KUKA KRL program: Safety_Position.src, Safety_Position.dat

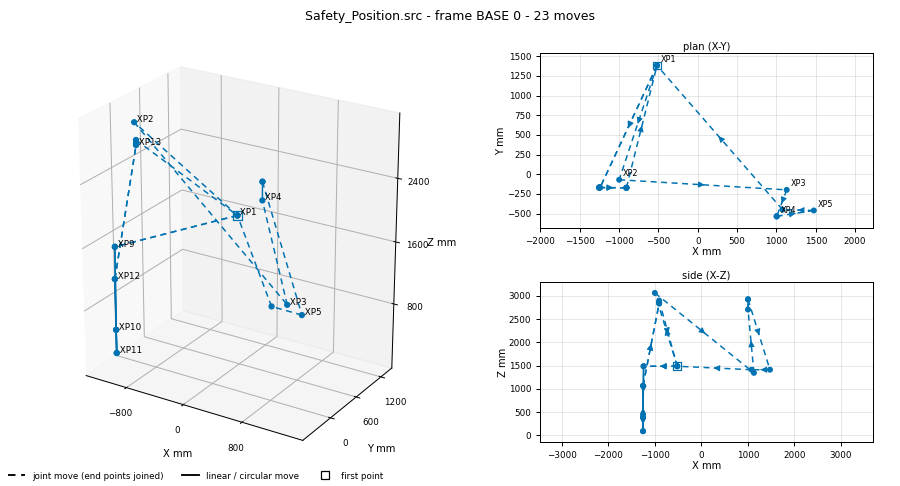
[picture p0: tool path of Safety_Position.src in frame BASE 0, 23 of 23 moves have a stored position in this frame; points joined in program order, loops and branches not executed]
--- Safety_Position.src ---
&ACCESS RVP8
&REL 86
&COMMENT Safety Position
&PARAM DISKPATH = KRC:\R1\Program\Safety Programs
DEF SAFETY_POSITION(DIRECTION :IN,AREA_NR :IN,TYPE_NR :IN )
;FOLD INI
  INT DIRECTION
  INT AREA_NR
  INT TYPE_NR
  decl KrlMsg_T msg
  decl KrlMsgPar_T par[3]
  decl KrlMsgOpt_T opt
  INT nHandle

  IF (DIRECTION>2) OR (DIRECTION<1) THEN
    REPEAT
      msg = {modul[] "Safety Position", nr 1, msg_txt[] "Direction Number Not Valid"}

			opt = {vl_stop true, clear_p_reset true, clear_p_SAW false, log_to_DB false}

			nHandle = Set_KrlMsg(#notify, msg, par[], opt)
      HALT
    UNTIL (DIRECTION<3) AND (DIRECTION>0)
  ENDIF
  IF (AREA_NR>8) OR (AREA_NR<1) THEN
    REPEAT
      msg = {modul[] "Safety Position", nr 2, msg_txt[] "Area Number Not Valid"}

			opt = {vl_stop true, clear_p_reset true, clear_p_SAW false, log_to_DB false}

			nHandle = Set_KrlMsg(#notify, msg, par[], opt)
      HALT
    UNTIL (AREA_NR<9) AND (AREA_NR>0)
  ENDIF
  IF (TYPE_NR>8) OR (TYPE_NR<1) THEN
    REPEAT
  	  msg = {modul[] "Safety Position", nr 1, msg_txt[] "Type Number Not Valid"}

			opt = {vl_stop true, clear_p_reset true, clear_p_SAW false, log_to_DB false}

			nHandle = Set_KrlMsg(#notify, msg, par[], opt)
      HALT
    UNTIL (TYPE_NR<9) AND (TYPE_NR>0)
  ENDIF
  ;ENDFOLD
;===================================================
; MODEL     :CX482
; IE GROUP  :PHEV
; STATION   :110
; ROBOT     :110R1
; FUNCTION  : Safety Position
;================================================

SWITCH AREA_NR

CASE 1  ;AREA 1

  SWITCH TYPE_NR

  CASE 1  ;Area 1 - Safety Position 1
    SWITCH DIRECTION
    CASE 1
    ;Teach here positions from wait area to safety position
;FOLD PTP P1 CONT Vel=50 % PDAT1 Tool[5] Base[0];%{PE}%R 8.3.48,%MKUKATPBASIS,%CMOVE,%VPTP,%P 1:PTP, 2:P1, 3:C_DIS, 5:50, 7:PDAT1
$BWDSTART=FALSE
PDAT_ACT=PPDAT1
FDAT_ACT=FP1
BAS(#PTP_PARAMS,50)
PTP XP1 C_DIS
;ENDFOLD
;FOLD PTP P2 Vel=50 % PDAT2 Tool[5] Base[0];%{PE}%R 8.3.48,%MKUKATPBASIS,%CMOVE,%VPTP,%P 1:PTP, 2:P2, 3:, 5:50, 7:PDAT2
$BWDSTART=FALSE
PDAT_ACT=PPDAT2
FDAT_ACT=FP2
BAS(#PTP_PARAMS,50)
PTP XP2
;ENDFOLD
    ;check robot movement for collision with other robots
    CASE 2
    ;Teach here positions from safety position to wait area
;FOLD PTP P3 CONT Vel=100 % PDAT3 Tool[5] Base[0];%{PE}%R 8.3.48,%MKUKATPBASIS,%CMOVE,%VPTP,%P 1:PTP, 2:P3, 3:C_DIS, 5:100, 7:PDAT3
$BWDSTART=FALSE
PDAT_ACT=PPDAT3
FDAT_ACT=FP3
BAS(#PTP_PARAMS,100)
PTP XP3 C_DIS
;ENDFOLD
;FOLD PTP P4 Vel=100 % PDAT4 Tool[5] Base[0];%{PE}%R 8.3.48,%MKUKATPBASIS,%CMOVE,%VPTP,%P 1:PTP, 2:P4, 3:, 5:100, 7:PDAT4
$BWDSTART=FALSE
PDAT_ACT=PPDAT4
FDAT_ACT=FP4
BAS(#PTP_PARAMS,100)
PTP XP4
;ENDFOLD
    ;check robot movement for collision with other robots
    ENDSWITCH

  CASE 2  ;Area 1 - Safety Position 2

    SWITCH DIRECTION
    CASE 1
lin_rel {z 220}
lin_rel {b 20}
;FOLD PTP P5 CONT Vel=100 % PDAT5 Tool[5] Base[0];%{PE}%R 8.3.48,%MKUKATPBASIS,%CMOVE,%VPTP,%P 1:PTP, 2:P5, 3:C_DIS, 5:100, 7:PDAT5
$BWDSTART=FALSE
PDAT_ACT=PPDAT5
FDAT_ACT=FP5
BAS(#PTP_PARAMS,100)
PTP XP5 C_DIS
;ENDFOLD
;FOLD PTP P7 CONT Vel=100 % PDAT7 Tool[5] Base[0];%{PE}%R 8.3.48,%MKUKATPBASIS,%CMOVE,%VPTP,%P 1:PTP, 2:P7, 3:C_DIS, 5:100, 7:PDAT7
$BWDSTART=FALSE
PDAT_ACT=PPDAT7
FDAT_ACT=FP7
BAS(#PTP_PARAMS,100)
PTP XP7 C_DIS
;ENDFOLD
;FOLD PTP P6 CONT Vel=100 % PDAT6 Tool[5] Base[0];%{PE}%R 8.3.48,%MKUKATPBASIS,%CMOVE,%VPTP,%P 1:PTP, 2:P6, 3:C_DIS, 5:100, 7:PDAT6
$BWDSTART=FALSE
PDAT_ACT=PPDAT6
FDAT_ACT=FP6
BAS(#PTP_PARAMS,100)
PTP XP6 C_DIS
;ENDFOLD
;FOLD PTP P9 CONT Vel=100 % PDAT9 Tool[5] Base[0];%{PE}%R 8.3.48,%MKUKATPBASIS,%CMOVE,%VPTP,%P 1:PTP, 2:P9, 3:C_DIS, 5:100, 7:PDAT9
$BWDSTART=FALSE
PDAT_ACT=PPDAT9
FDAT_ACT=FP9
BAS(#PTP_PARAMS,100)
PTP XP9 C_DIS
;ENDFOLD
;FOLD LIN P10 CONT Vel=2 m/s CPDAT1 Tool[5] Base[0];%{PE}%R 8.3.48,%MKUKATPBASIS,%CMOVE,%VLIN,%P 1:LIN, 2:P10, 3:C_DIS C_DIS, 5:2, 7:CPDAT1
$BWDSTART=FALSE
LDAT_ACT=LCPDAT1
FDAT_ACT=FP10
BAS(#CP_PARAMS,2)
LIN XP10 C_DIS C_DIS
;ENDFOLD
;FOLD LIN P11 Vel=0.5 m/s CPDAT2 Tool[5] Base[0];%{PE}%R 8.3.48,%MKUKATPBASIS,%CMOVE,%VLIN,%P 1:LIN, 2:P11, 3:, 5:0.5, 7:CPDAT2
$BWDSTART=FALSE
LDAT_ACT=LCPDAT2
FDAT_ACT=FP11
BAS(#CP_PARAMS,0.5)
LIN XP11
;ENDFOLD

;abrir gara
cil_bat_reposo()

;FOLD LIN P12 CONT Vel=0.5 m/s CPDAT3 Tool[5] Base[0];%{PE}%R 8.3.48,%MKUKATPBASIS,%CMOVE,%VLIN,%P 1:LIN, 2:P12, 3:C_DIS C_DIS, 5:0.5, 7:CPDAT3
$BWDSTART=FALSE
LDAT_ACT=LCPDAT3
FDAT_ACT=FP12
BAS(#CP_PARAMS,0.5)
LIN XP12 C_DIS C_DIS
;ENDFOLD
;FOLD PTP P13 CONT Vel=100 % PDAT10 Tool[5] Base[0];%{PE}%R 8.3.48,%MKUKATPBASIS,%CMOVE,%VPTP,%P 1:PTP, 2:P13, 3:C_DIS, 5:100, 7:PDAT10
$BWDSTART=FALSE
PDAT_ACT=PPDAT10
FDAT_ACT=FP13
BAS(#PTP_PARAMS,100)
PTP XP13 C_DIS
;ENDFOLD
    ;Teach here positions from waiting area to safety position
    ;check robot movement for collision with other robots
    CASE 2
lin_rel {z 20}
lin_rel {b 20}
lin_rel {z 40}
;FOLD PTP P14 CONT Vel=100 % PDAT11 Tool[5] Base[0];%{PE}%R 8.3.48,%MKUKATPBASIS,%CMOVE,%VPTP,%P 1:PTP, 2:P14, 3:C_DIS, 5:100, 7:PDAT11
$BWDSTART=FALSE
PDAT_ACT=PPDAT11
FDAT_ACT=FP14
BAS(#PTP_PARAMS,100)
PTP XP14 C_DIS
;ENDFOLD
;FOLD PTP P15 CONT Vel=100 % PDAT12 Tool[5] Base[0];%{PE}%R 8.3.48,%MKUKATPBASIS,%CMOVE,%VPTP,%P 1:PTP, 2:P15, 3:C_DIS, 5:100, 7:PDAT12
$BWDSTART=FALSE
PDAT_ACT=PPDAT12
FDAT_ACT=FP15
BAS(#PTP_PARAMS,100)
PTP XP15 C_DIS
;ENDFOLD
;FOLD LIN P16 CONT Vel=0.5 m/s CPDAT4 Tool[5] Base[0];%{PE}%R 8.3.48,%MKUKATPBASIS,%CMOVE,%VLIN,%P 1:LIN, 2:P16, 3:C_DIS C_DIS, 5:0.5, 7:CPDAT4
$BWDSTART=FALSE
LDAT_ACT=LCPDAT4
FDAT_ACT=FP16
BAS(#CP_PARAMS,0.5)
LIN XP16 C_DIS C_DIS
;ENDFOLD
;FOLD LIN P17 Vel=0.5 m/s CPDAT5 Tool[5] Base[0];%{PE}%R 8.3.48,%MKUKATPBASIS,%CMOVE,%VLIN,%P 1:LIN, 2:P17, 3:, 5:0.5, 7:CPDAT5
$BWDSTART=FALSE
LDAT_ACT=LCPDAT5
FDAT_ACT=FP17
BAS(#CP_PARAMS,0.5)
LIN XP17
;ENDFOLD

;abrir gara
cil_bat_reposo()

;FOLD LIN P18 CONT Vel=0.5 m/s CPDAT6 Tool[5] Base[0];%{PE}%R 8.3.48,%MKUKATPBASIS,%CMOVE,%VLIN,%P 1:LIN, 2:P18, 3:C_DIS C_DIS, 5:0.5, 7:CPDAT6
$BWDSTART=FALSE
LDAT_ACT=LCPDAT6
FDAT_ACT=FP18
BAS(#CP_PARAMS,0.5)
LIN XP18 C_DIS C_DIS
;ENDFOLD
;FOLD PTP P19 CONT Vel=100 % PDAT13 Tool[5] Base[0];%{PE}%R 8.3.48,%MKUKATPBASIS,%CMOVE,%VPTP,%P 1:PTP, 2:P19, 3:C_DIS, 5:100, 7:PDAT13
$BWDSTART=FALSE
PDAT_ACT=PPDAT13
FDAT_ACT=FP19
BAS(#PTP_PARAMS,100)
PTP XP19 C_DIS
;ENDFOLD
    ;Teach here positions from safety position to waiting area
    ;check robot movement for collision with other robots
    ENDSWITCH

  CASE 3  ;Area 1 - Safety Position 3

    SWITCH DIRECTION
    CASE 1
    ;Teach here positions from waiting area to safety position
    ;check robot movement for collision with other robots
    CASE 2
    ;Teach here positions from safety position to waiting area
    ;check robot movement for collision with other robots
    ENDSWITCH

  CASE 4  ;Area 1 - Safety Position 4

    SWITCH DIRECTION
    CASE 1 ; From Area Request Position To Safety Position
    ;Teach here positions from waiting area to safety position
    ;check robot movement for collision with other robots
    CASE 2 ; From Safety Position To Area Request Position
    ;Teach here positions from safety position to waiting area
    ;check robot movement for collision with other robots
    ENDSWITCH

  CASE 5  ;Area 1 - Safety Position 5

    SWITCH DIRECTION
    CASE 1
    ;Teach here positions from waiting area to safety position
    ;check robot movement for collision with other robots
    CASE 2
    ;Teach here positions from safety position to waiting area
    ;check robot movement for collision with other robots
    ENDSWITCH

  CASE 6  ;Area 1 - Safety Position 6

    SWITCH DIRECTION
    CASE 1
    ;Teach here positions from waiting area to safety position
    ;check robot movement for collision with other robots
    CASE 2
    ;Teach here positions from safety position to waiting area
    ;check robot movement for collision with other robots
    ENDSWITCH

  CASE 7  ;Area 1 - Safety Position 7

    SWITCH DIRECTION
    CASE 1
    ;Teach here positions from waiting area to safety position
    ;check robot movement for collision with other robots
    CASE 2
    ;Teach here positions from safety position to waiting area
    ;check robot movement for collision with other robots
    ENDSWITCH

  CASE 8  ;Area 1 - Safety Position 8

    SWITCH DIRECTION
    CASE 1
    ;Teach here positions from wait area to safety position
    ;check robot movement for collision with other robots
    CASE 2
    ;Teach here positions from safety position to wait area
    ;check robot movement for collision with other robots
    ENDSWITCH

  ENDSWITCH

;====================================================================

CASE 2  ;AREA 2

  SWITCH TYPE_NR
  CASE 1  ;Area 2 - Safety Position 1

    SWITCH DIRECTION
    CASE 1
    ;Teach here pos from waiting area to safety position
    ;check robot movement for collision with other robots
    CASE 2
    ;Teach here positions from safety pos to waiting area
    ;check robot movement for collision with other robots
    ENDSWITCH

  CASE 2  ;Area 2 - Safety Position 2

    SWITCH DIRECTION
    CASE 1
    ;Teach here positions from waiting area to safety position
    ;check robot movement for collision with other robots
    CASE 2
    ;Teach here positions from safety position to waiting area
    ;check robot movement for collision with other robots
    ENDSWITCH

  CASE 3  ;Area 2 - Safety Position 3

    SWITCH DIRECTION
    CASE 1
    ;Teach here positions from waiting area to safety position
    ;check robot movement for collision with other robots
    CASE 2
    ;Teach here positions from safety position to waiting area
    ;check robot movement for collision with other robots
    ENDSWITCH

  CASE 4  ;Area 2 - Safety Position 4

    SWITCH DIRECTION
	  	CASE 1
    ;Teach here positions from waiting area to safety position
    ;check robot movement for collision with other robots
    CASE 2
    ;Teach here positions from safety position to waiting area
    ;check robot movement for collision with other robots
    ENDSWITCH

  CASE 5  ;Area 2 - Safety Position 5

    SWITCH DIRECTION
    CASE 1
    ;Teach here positions from waiting area to safety position
    ;check robot movement for collision with other robots
    CASE 2
    ;Teach here positions from safety position to waiting area
    ;check robot movement for collision with other robots
    ENDSWITCH

  CASE 6    ;Area 2 - Safety Position 6

    SWITCH DIRECTION
    CASE 1
    ;Teach here positions from waiting area to safety position
    ;check robot movement for collision with other robots
    CASE 2
    ;Teach here positions from safety position to waiting area
    ;check robot movement for collision with other robots
    ENDSWITCH

  CASE 7    ;Area 2 - Safety Position 7

    SWITCH DIRECTION
    CASE 1
    ;Teach here positions from waiting area to safety position
    ;check robot movement for collision with other robots
    CASE 2
    ;Teach here positions from safety position to waiting area
    ;check robot movement for collision with other robots
    ENDSWITCH

  CASE 8  ;Area 2 - Safety Position 8

    SWITCH DIRECTION
    CASE 1
    ;Teach here positions from waiting area to safety position
    ;check robot movement for collision with other robots
    CASE 2
    ;Teach here positions from safety position to waiting area
    ;check robot movement for collision with other robots
    ENDSWITCH

  ENDSWITCH

;====================================================================

CASE 3  ;AREA 3

  SWITCH TYPE_NR
  CASE 1  ;Area 3 - Safety Position 1

    SWITCH DIRECTION
    CASE 1
    ;Teach here positions from waiting area to safety position
    ;check robot movement for collision with other robots
    CASE 2
    ;Teach here positions from safety position to waiting area
    ;check robot movement for collision with other robots
    ENDSWITCH

  CASE 2  ;Area 3 - Safety Position 2

    SWITCH DIRECTION
    CASE 1
    ;Teach here positions from waiting area to safety position
    ;check robot movement for collision with other robots
    CASE 2
    ;Teach here positions from safety position to waiting area
    ;check robot movement for collision with other robots
    ENDSWITCH

  CASE 3  ;Area 3 - Safety Position 3

    SWITCH DIRECTION
    CASE 1
    ;Teach here positions from waiting area to safety position
    ;check robot movement for collision with other robots
    CASE 2
    ;Teach here positions from safety position to waiting area
    ;check robot movement for collision with other robots
      ENDSWITCH

  CASE 4  ;Area 3 - Safety Position 4

    SWITCH DIRECTION
    CASE 1
    ;Teach here positions from waiting area to safety position
    ;check robot movement for collision with other robots
    CASE 2
    ;Teach here positions from safety position to waiting area
    ;check robot movement for collision with other robots
    ENDSWITCH

  CASE 5  ;Area 3 - Safety Position 5

    SWITCH DIRECTION
    CASE 1
    ;Teach here positions from waiting area to safety position
    ;check robot movement for collision with other robots
    CASE 2
    ;Teach here positions from safety position to waiting area
    ;check robot movement for collision with other robots
    ENDSWITCH

  CASE 6  ;Area 3 - Safety Position 6

    SWITCH DIRECTION
    CASE 1
    ;Teach here positions from waiting area to safety position
    ;check robot movement for collision with other robots
    CASE 2
    ;Teach here positions from safety position to waiting area
    ;check robot movement for collision with other robots
    ENDSWITCH

  CASE 7  ;Area 3 - Safety Position 7

    SWITCH DIRECTION
    CASE 1
    ;Teach here positions from waiting area to safety position
    ;check robot movement for collision with other robots
    CASE 2
    ;Teach here positions from safety position to waiting area
    ;check robot movement for collision with other robots
    ENDSWITCH

  CASE 8  ;Area 3 - Safety Position 8
    SWITCH DIRECTION
    CASE 1
    ;Teach here positions from waiting area to safety position
    ;check robot movement for collision with other robots
    CASE 2
    ;Teach here positions from safety position to waiting area
    ;check robot movement for collision with other robots
    ENDSWITCH

  ENDSWITCH

;====================================================================

CASE 4  ;AREA 4

  SWITCH TYPE_NR
  CASE 1  ;Area 4 - Safety Position 1

    SWITCH DIRECTION
    CASE 1
		;Teach here positions from waiting area to safety position
		;check robot movement for collision with other robots
		CASE 2
		;Teach here positions from safety position to waiting area
		;check robot movement for collision with other robots

    ENDSWITCH

  CASE 2  ;Area 4 - Safety Position 2

    SWITCH DIRECTION
    CASE 1
	  ;Teach here positions from waiting area to safety position
	  ;check robot movement for collision with other robots
    CASE 2
	  ;Teach here positions from safety position to waiting area
  	;check robot movement for collision with other robots
    ENDSWITCH

  CASE 3  ;Area 4 - Safety Position 3

    SWITCH DIRECTION
    CASE 1
    ;Teach here positions from waiting area to safety position
    ;check robot movement for collision with other robots
    CASE 2
    ;Teach here positions from safety position to waiting area
    ;check robot movement for collision with other robots
    ENDSWITCH

  CASE 4  ;Area 4 - Safety Position 4

    SWITCH DIRECTION
    CASE 1
    ;Teach here positions from waiting area to safety position
    ;check robot movement for collision with other robots
    CASE 2
    ;Teach here positions from safety position to waiting area
    ;check robot movement for collision with other robots
    ENDSWITCH

  CASE 5  ;Area 4 - Safety Position 5

    SWITCH DIRECTION
    CASE 1
    ;Teach here positions from waiting area to safety position
    ;check robot movement for collision with other robots
    CASE 2
    ;Teach here positions from safety position to waiting area
    ;check robot movement for collision with other robots
    ENDSWITCH

  CASE 6  ;Area 4 - Safety Position 6

    SWITCH DIRECTION
    CASE 1
    ;Teach here positions from waiting area to safety position
    ;check robot movement for collision with other robots
    CASE 2
    ;Teach here positions from safety position to waiting area
    ;check robot movement for collision with other robots
    ENDSWITCH

  CASE 7  ;Area 4 - Safety Position 7

    SWITCH DIRECTION
    CASE 1
    ;Teach here positions from waiting area to safety position
    ;check robot movement for collision with other robots
    CASE 2
    ;Teach here positions from safety position to waiting area
    ;check robot movement for collision with other robots
    ENDSWITCH

  CASE 8  ;Area 4 - Safety Position 8

    SWITCH DIRECTION
    CASE 1
    ;Teach here positions from waiting area to safety position
    ;check robot movement for collision with other robots
    CASE 2
    ;Teach here positions from safety position to waiting area
    ;check robot movement for collision with other robots
    ENDSWITCH

  ENDSWITCH

;====================================================================

CASE 5  ;AREA 5

  SWITCH TYPE_NR
  CASE 1  ;Area 5 - Safety Position 1

    SWITCH DIRECTION
    CASE 1
    ;Teach here positions from waiting area to safety position
    ;check robot movement for collision with other robots
    CASE 2
    ;Teach here positions from safety position to waiting area
    ;check robot movement for collision with other robots
    ENDSWITCH

  CASE 2  ;Area 5 - Safety Position 2

    SWITCH DIRECTION
    CASE 1
    ;Teach here positions from waiting area to safety position
    ;check robot movement for collision with other robots
    CASE 2
    ;Teach here positions from safety position to waiting area
    ;check robot movement for collision with other robots
    ENDSWITCH

  CASE 3  ;Area 5 - Safety Position 3

    SWITCH DIRECTION
    CASE 1
    ;Teach here positions from waiting area to safety position
    ;check robot movement for collision with other robots
    CASE 2
    ;Teach here positions from safety position to waiting area
    ;check robot movement for collision with other robots
    ENDSWITCH

  CASE 4  ;Area 5 - Safety Position 4

    SWITCH DIRECTION
    CASE 1
    ;Teach here positions from waiting area to safety position
    ;check robot movement for collision with other robots
    CASE 2
    ;Teach here positions from safety position to waiting area
    ;check robot movement for collision with other robots
    ENDSWITCH

  CASE 5  ;Area 5 - Safety Position 5

    SWITCH DIRECTION
    CASE 1
    ;Teach here positions from waiting area to safety position
    ;check robot movement for collision with other robots
    CASE 2
    ;Teach here positions from safety position to waiting area
    ;check robot movement for collision with other robots
    ENDSWITCH

  CASE 6  ;Area 5 - Safety Position 6

    SWITCH DIRECTION
    CASE 1
    ;Teach here positions from waiting area to safety position
    ;check robot movement for collision with other robots
    CASE 2
    ;Teach here positions from safety position to waiting area
    ;check robot movement for collision with other robots
    ENDSWITCH

  CASE 7  ;Area 5 - Safety Position 7

    SWITCH DIRECTION
    CASE 1
    ;Teach here positions from waiting area to safety position
    ;check robot movement for collision with other robots
    CASE 2
    ;Teach here positions from safety position to waiting area
    ;check robot movement for collision with other robots
    ENDSWITCH

  CASE 8  ;Area 5 - Safety Position 8

    SWITCH DIRECTION
    CASE 1
    ;Teach here positions from waiting area to safety position
    ;check robot movement for collision with other robots
    CASE 2
    ;Teach here positions from safety position to waiting area
    ;check robot movement for collision with other robots
    ENDSWITCH

  ENDSWITCH

;====================================================================

CASE 6  ;AREA 6

  SWITCH TYPE_NR
  CASE 1  ;Area 6 - Safety Position 1

    SWITCH DIRECTION
    CASE 1
    ;Teach here positions from waiting area to safety position
    ;check robot movement for collision with other robots
    CASE 2
    ;Teach here positions from safety position to waiting area
    ;check robot movement for collision with other robots
    ENDSWITCH

  CASE 2  ;Area 6 - Safety Position 2

    SWITCH DIRECTION
    CASE 1
    ;Teach here positions from waiting area to safety position
    ;check robot movement for collision with other robots
    CASE 2
    ;Teach here positions from safety position to waiting area
    ;check robot movement for collision with other robots
    ENDSWITCH

  CASE 3  ;Area 6 - Safety Position 3

    SWITCH DIRECTION
    CASE 1
    ;Teach here positions from waiting area to safety position
    ;check robot movement for collision with other robots
    CASE 2
    ;Teach here positions from safety position to waiting area
    ;check robot movement for collision with other robots
    ENDSWITCH

  CASE 4  ;Area 6 - Safety Position 4

    SWITCH DIRECTION
    CASE 1
    ;Teach here positions from waiting area to safety position
    ;check robot movement for collision with other robots
    CASE 2
    ;Teach here positions from safety position to waiting area
    ;check robot movement for collision with other robots
    ENDSWITCH

  CASE 5  ;Area 6 - Safety Position 5

    SWITCH DIRECTION
    CASE 1
    ;Teach here positions from waiting area to safety position
    ;check robot movement for collision with other robots
    CASE 2
    ;Teach here positions from safety position to waiting area
    ;check robot movement for collision with other robots
    ENDSWITCH

  CASE 6  ;Area 6 - Safety Position 6

    SWITCH DIRECTION
    CASE 1
    ;Teach here positions from waiting area to safety position
    ;check robot movement for collision with other robots
    CASE 2
    ;Teach here positions from safety position to waiting area
    ;check robot movement for collision with other robots
    ENDSWITCH

  CASE 7  ;Area 6 - Safety Position 7

    SWITCH DIRECTION
    CASE 1
    ;Teach here positions from waiting area to safety position
    ;check robot movement for collision with other robots
    CASE 2
    ;Teach here positions from safety position to waiting area
    ;check robot movement for collision with other robots
    ENDSWITCH

  CASE 8  ;Area 6 - Safety Position 8

    SWITCH DIRECTION
    CASE 1
    ;Teach here positions from waiting area to safety position
    ;check robot movement for collision with other robots
    CASE 2
    ;Teach here positions from safety position to waiting area
    ;check robot movement for collision with other robots
    ENDSWITCH

  ENDSWITCH

;====================================================================

CASE 7  ;AREA 7

  SWITCH TYPE_NR
  CASE 1  ;Area 7 - Safety Position 1

    SWITCH DIRECTION
    CASE 1
    ;Teach here positions from waiting area to safety position
    ;check robot movement for collision with other robots
    CASE 2
    ;Teach here positions from safety position to waiting area
    ;check robot movement for collision with other robots
    ENDSWITCH

  CASE 2  ;Area 7 - Safety Position 2

    SWITCH DIRECTION
    CASE 1
    ;Teach here positions from waiting area to safety position
    ;check robot movement for collision with other robots
    CASE 2
    ;Teach here positions from safety position to waiting area
    ;check robot movement for collision with other robots
    ENDSWITCH

  CASE 3  ;Area 7 - Safety Position 3

    SWITCH DIRECTION
    CASE 1
    ;Teach here positions from waiting area to safety position
    ;check robot movement for collision with other robots
    CASE 2
    ;Teach here positions from safety position to waiting area
    ;check robot movement for collision with other robots
    ENDSWITCH

  CASE 4  ;Area 7 - Safety Position 4

    SWITCH DIRECTION
    CASE 1
    ;Teach here positions from waiting area to safety position
    ;check robot movement for collision with other robots
    CASE 2
    ;Teach here positions from safety position to waiting area
    ;check robot movement for collision with other robots
    ENDSWITCH

  CASE 5  ;Area 7 - Safety Position 5

    SWITCH DIRECTION
    CASE 1
    ;Teach here positions from waiting area to safety position
    ;check robot movement for collision with other robots
    CASE 2
    ;Teach here positions from safety position to waiting area
    ;check robot movement for collision with other robots
    ENDSWITCH

  CASE 6  ;Area 7 - Safety Position 6

    SWITCH DIRECTION
    CASE 1
    ;Teach here positions from waiting area to safety position
    ;check robot movement for collision with other robots
    CASE 2
    ;Teach here positions from safety position to waiting area
    ;check robot movement for collision with other robots
    ENDSWITCH

  CASE 7  ;Area 7 - Safety Position 7

    SWITCH DIRECTION
    CASE 1
    ;Teach here positions from waiting area to safety position
    ;check robot movement for collision with other robots
    CASE 2
    ;Teach here positions from safety position to waiting area
    ;check robot movement for collision with other robots
    ENDSWITCH

  CASE 8  ;Area 7 - Safety Position 8

    SWITCH DIRECTION
    CASE 1
    ;Teach here positions from waiting area to safety position
    ;check robot movement for collision with other robots
    CASE 2
    ;Teach here positions from safety position to waiting area
    ;check robot movement for collision with other robots
    ENDSWITCH

  ENDSWITCH

;====================================================================

CASE 8  ;AREA 8

  SWITCH TYPE_NR
  CASE 1  ;Area 8 - Safety Position 1

    SWITCH DIRECTION
    CASE 1
    ;Teach here positions from waiting area to safety position
    ;check robot movement for collision with other robots
    CASE 2
    ;Teach here positions from safety position to waiting area
    ;check robot movement for collision with other robots
    ENDSWITCH

  CASE 2  ;Area 8 - Safety Position 2

    SWITCH DIRECTION
    CASE 1
    ;Teach here positions from waiting area to safety position
    ;check robot movement for collision with other robots
    CASE 2
    ;Teach here positions from safety position to waiting area
    ;check robot movement for collision with other robots
    ENDSWITCH

  CASE 3  ;Area 8 - Safety Position 3

    SWITCH DIRECTION
    CASE 1
    ;Teach here positions from waiting area to safety position
    ;check robot movement for collision with other robots
    CASE 2
    ;Teach here positions from safety position to waiting area
    ;check robot movement for collision with other robots
    ENDSWITCH

  CASE 4  ;Area 8 - Safety Position 4

    SWITCH DIRECTION
    CASE 1
    ;Teach here positions from waiting area to safety position
    ;check robot movement for collision with other robots
    CASE 2
    ;Teach here positions from safety position to waiting area
    ;check robot movement for collision with other robots
    ENDSWITCH

  CASE 5  ;Area 8 - Safety Position 5

    SWITCH DIRECTION
    CASE 1
    ;Teach here positions from waiting area to safety position
    ;check robot movement for collision with other robots
    CASE 2
    ;Teach here positions from safety position to waiting area
    ;check robot movement for collision with other robots
    ENDSWITCH

  CASE 6  ;Area 8 - Safety Position 6

    SWITCH DIRECTION
    CASE 1
    ;Teach here positions from waiting area to safety position
    ;check robot movement for collision with other robots
    CASE 2
    ;Teach here positions from safety position to waiting area
    ;check robot movement for collision with other robots
    ENDSWITCH

  CASE 7  ;Area 8 - Safety Position 7

    SWITCH DIRECTION
    CASE 1
    ;Teach here positions from waiting area to safety position
    ;check robot movement for collision with other robots
    CASE 2
    ;Teach here positions from safety position to waiting area
    ;check robot movement for collision with other robots
    ENDSWITCH

  CASE 8  ;Area 8 - Safety Position 8

    SWITCH DIRECTION
    CASE 1
    ;Teach here positions from waiting area to safety position
    ;check robot movement for collision with other robots
    CASE 2
    ;Teach here positions from safety position to waiting area
    ;check robot movement for collision with other robots
    ENDSWITCH
  ENDSWITCH
ENDSWITCH
END

--- Safety_Position.dat ---
&ACCESS RVP8
&REL 86
&COMMENT Safety Position
&PARAM DISKPATH = KRC:\R1\Program\Safety Programs
DEFDAT  Safety_Position
;FOLD EXTERNAL DECLARATIONS;%{PE}%V3.2.0,%MKUKATPBASIS,%CEXT,%VCOMMON,%P
;FOLD BAS EXT;%{PE}%V3.2.0,%MKUKATPBASIS,%CEXT,%VEXT,%P
EXT  BAS (BAS_COMMAND  :IN,REAL  :IN )
DECL INT SUCCESS
;ENDFOLD
;FOLD GRIPPERTECH EXT
EXT  H50 (INT  :IN,INT  :IN,INT  :IN,GRP_TYP  :IN )
;ENDFOLD (GRIPPERTECH EXT)
;FOLD SPOTTECH EXT
EXT  USERSPOT (S_COMMAND  :IN,SPOT_TYPE  :IN )
;ENDFOLD (SPOTTECH EXT)
;FOLD USER EXT;%{E}%V3.2.0,%MKUKATPUSER,%CEXT,%VEXT,%P
;Make here your modifications
;ENDFOLD
;ENDFOLD

DECL E6POS XP1={X -517.192932,Y 1381.33044,Z 1487.17358,A -88.9551926,B 22.2455845,C 175.857315,S 6,T 27,E1 0.0,E2 0.0,E3 0.0,E4 0.0,E5 0.0,E6 0.0}
DECL BASIS_SUGG_T LAST_BASIS={POINT1[] "P19                     ",POINT2[] "P19                     ",CP_PARAMS[] "CPDAT6                  ",PTP_PARAMS[] "PDAT13                  ",CONT[] "C_DIS                   ",CP_VEL[] "0.5                     ",PTP_VEL[] "100                     ",SYNC_PARAMS[] "SYNCDAT                 ",SPL_NAME[] "S0                      ",A_PARAMS[] "ADAT0                   "}
DECL FDAT FP1={TOOL_NO 5,BASE_NO 0,IPO_FRAME #BASE,POINT2[] " ",TQ_STATE FALSE}
DECL PDAT PPDAT1={VEL 100.000,ACC 100.000,APO_DIST 100.000,APO_MODE #CDIS,GEAR_JERK 50.0000,EXAX_IGN 0}
DECL E6POS XP2={X -997.814392,Y -69.8441467,Z 3061.98706,A -167.261963,B 53.2046585,C 15.6102886,S 6,T 27,E1 0.0,E2 0.0,E3 0.0,E4 0.0,E5 0.0,E6 0.0}
DECL FDAT FP2={TOOL_NO 5,BASE_NO 0,IPO_FRAME #BASE,POINT2[] " ",TQ_STATE FALSE}
DECL PDAT PPDAT2={VEL 100.000,ACC 100.000,APO_DIST 100.000,GEAR_JERK 50.0000,EXAX_IGN 0}
DECL E6POS XP3={X 1130.65405,Y -198.428650,Z 1344.54492,A -170.437561,B 0.776786268,C 179.869324,S 6,T 26,E1 0.0,E2 0.0,E3 0.0,E4 0.0,E5 0.0,E6 0.0}
DECL FDAT FP3={TOOL_NO 5,BASE_NO 0,IPO_FRAME #BASE,POINT2[] " ",TQ_STATE FALSE}
DECL PDAT PPDAT3={VEL 100.000,ACC 100.000,APO_DIST 100.000,APO_MODE #CDIS,GEAR_JERK 50.0000,EXAX_IGN 0}
DECL E6POS XP4={X 1003.54260,Y -534.980896,Z 2705.33,A 46.6126213,B 2.57036543,C 13.6730404,S 2,T 10,E1 0.0,E2 0.0,E3 0.0,E4 0.0,E5 0.0,E6 0.0}
DECL FDAT FP4={TOOL_NO 5,BASE_NO 0,IPO_FRAME #BASE,POINT2[] " ",TQ_STATE FALSE}
DECL PDAT PPDAT4={VEL 100.000,ACC 100.000,APO_DIST 100.000,GEAR_JERK 50.0000,EXAX_IGN 0}
DECL E6POS XP5={X 1475.14294,Y -460.159363,Z 1412.20422,A -177.899490,B 3.32464623,C -176.200607,S 6,T 26,E1 0.0,E2 0.0,E3 0.0,E4 0.0,E5 0.0,E6 0.0}
DECL FDAT FP5={TOOL_NO 5,BASE_NO 0,IPO_FRAME #BASE,POINT2[] " ",TQ_STATE FALSE}
DECL PDAT PPDAT5={VEL 100.000,ACC 100.000,APO_DIST 100.000,APO_MODE #CDIS,GEAR_JERK 50.0000,EXAX_IGN 0}
DECL E6POS XP6={X -517.192932,Y 1381.33044,Z 1487.17358,A -88.9551926,B 22.2455845,C 175.857315,S 6,T 27,E1 0.0,E2 0.0,E3 0.0,E4 0.0,E5 0.0,E6 0.0}
DECL FDAT FP6={TOOL_NO 5,BASE_NO 0,IPO_FRAME #BASE,POINT2[] " ",TQ_STATE FALSE}
DECL PDAT PPDAT6={VEL 100.000,ACC 100.000,APO_DIST 100.000,APO_MODE #CDIS,GEAR_JERK 50.0000,EXAX_IGN 0}
DECL E6POS XP7={X 1076.88843,Y -449.355316,Z 1412.20129,A -177.899490,B 3.32450485,C -176.200607,S 6,T 26,E1 0.0,E2 0.0,E3 0.0,E4 0.0,E5 0.0,E6 0.0}
DECL FDAT FP7={TOOL_NO 5,BASE_NO 0,IPO_FRAME #BASE,POINT2[] " ",TQ_STATE FALSE}
DECL PDAT PPDAT7={VEL 100.000,ACC 100.000,APO_DIST 100.000,APO_MODE #CDIS,GEAR_JERK 50.0000,EXAX_IGN 0}
DECL E6POS XP8={X -1240.58252,Y -169.310059,Z 1486.69885,A -13.5853224,B 22.1978359,C 175.933182,S 6,T 27,E1 0.0,E2 0.0,E3 0.0,E4 0.0,E5 0.0,E6 0.0}
DECL FDAT FP8={TOOL_NO 5,BASE_NO 0,IPO_FRAME #BASE,POINT2[] " ",TQ_STATE FALSE}
DECL PDAT PPDAT8={VEL 100.000,ACC 100.000,APO_DIST 100.000,APO_MODE #CDIS,GEAR_JERK 50.0000,EXAX_IGN 0}
DECL E6POS XP9={X -1240.58252,Y -169.310059,Z 1486.69885,A -13.5853224,B 22.1978359,C 175.933182,S 6,T 27,E1 0.0,E2 0.0,E3 0.0,E4 0.0,E5 0.0,E6 0.0}
DECL FDAT FP9={TOOL_NO 5,BASE_NO 0,IPO_FRAME #BASE,POINT2[] " ",TQ_STATE FALSE}
DECL PDAT PPDAT9={VEL 100.000,ACC 100.000,APO_DIST 100.000,APO_MODE #CDIS,GEAR_JERK 50.0000,EXAX_IGN 0}
DECL E6POS XP10={X -1252.06714,Y -169.310547,Z 400.812317,A 0.119013771,B 2.16552854,C 179.742950,S 6,T 27,E1 0.0,E2 0.0,E3 0.0,E4 0.0,E5 0.0,E6 0.0}
DECL FDAT FP10={TOOL_NO 5,BASE_NO 0,IPO_FRAME #BASE,POINT2[] " ",TQ_STATE FALSE}
DECL LDAT LCPDAT1={VEL 2.00000,ACC 100.000,APO_DIST 100.000,APO_FAC 50.0000,AXIS_VEL 100.000,AXIS_ACC 100.000,ORI_TYP #VAR,CIRC_TYP #BASE,JERK_FAC 50.0000,GEAR_JERK 50.0000,EXAX_IGN 0}
DECL E6POS XP11={X -1252.07056,Y -169.310532,Z 91.2468262,A -1.23850,B 1.32794106,C 179.761078,S 6,T 27,E1 0.0,E2 0.0,E3 0.0,E4 0.0,E5 0.0,E6 0.0}
DECL FDAT FP11={TOOL_NO 5,BASE_NO 0,IPO_FRAME #BASE,POINT2[] " ",TQ_STATE FALSE}
DECL LDAT LCPDAT2={VEL 2.00000,ACC 100.000,APO_DIST 100.000,APO_FAC 50.0000,AXIS_VEL 100.000,AXIS_ACC 100.000,ORI_TYP #VAR,CIRC_TYP #BASE,JERK_FAC 50.0000,GEAR_JERK 50.0000,EXAX_IGN 0}
DECL E6POS XP12={X -1252.07043,Y -169.310532,Z 1067.28162,A -1.23849988,B 1.32794094,C 179.761078,S 6,T 27,E1 0.0,E2 0.0,E3 0.0,E4 0.0,E5 0.0,E6 0.0}
DECL FDAT FP12={TOOL_NO 5,BASE_NO 0,IPO_FRAME #BASE,POINT2[] " ",TQ_STATE FALSE}
DECL LDAT LCPDAT3={VEL 2.00000,ACC 100.000,APO_DIST 100.000,APO_FAC 50.0000,AXIS_VEL 100.000,AXIS_ACC 100.000,ORI_TYP #VAR,CIRC_TYP #BASE,JERK_FAC 50.0000,GEAR_JERK 50.0000,EXAX_IGN 0}
DECL E6POS XP13={X -905.921936,Y -172.186203,Z 2837.76685,A -5.97172117,B 82.0147247,C 174.335983,S 6,T 27,E1 0.0,E2 0.0,E3 0.0,E4 0.0,E5 0.0,E6 0.0}
DECL FDAT FP13={TOOL_NO 5,BASE_NO 0,IPO_FRAME #BASE,POINT2[] " ",TQ_STATE FALSE}
DECL PDAT PPDAT10={VEL 100.000,ACC 100.000,APO_DIST 100.000,APO_MODE #CDIS,GEAR_JERK 50.0000,EXAX_IGN 0}
DECL E6POS XP14={X -517.192932,Y 1381.33044,Z 1487.17358,A -88.9551926,B 22.2455845,C 175.857315,S 6,T 27,E1 0.0,E2 0.0,E3 0.0,E4 0.0,E5 0.0,E6 0.0}
DECL FDAT FP14={TOOL_NO 5,BASE_NO 0,IPO_FRAME #BASE,POINT2[] " ",TQ_STATE FALSE}
DECL PDAT PPDAT11={VEL 100.000,ACC 100.000,APO_DIST 100.000,APO_MODE #CDIS,GEAR_JERK 50.0000,EXAX_IGN 0}
DECL E6POS XP15={X -1240.58252,Y -169.310059,Z 1486.69885,A -13.5853224,B 22.1978359,C 175.933182,S 6,T 27,E1 0.0,E2 0.0,E3 0.0,E4 0.0,E5 0.0,E6 0.0}
DECL FDAT FP15={TOOL_NO 5,BASE_NO 0,IPO_FRAME #BASE,POINT2[] " ",TQ_STATE FALSE}
DECL PDAT PPDAT12={VEL 100.000,ACC 100.000,APO_DIST 100.000,APO_MODE #CDIS,GEAR_JERK 50.0000,EXAX_IGN 0}
DECL E6POS XP16={X -1252.06714,Y -169.310547,Z 400.812317,A 0.119013771,B 2.16552854,C 179.742950,S 6,T 27,E1 0.0,E2 0.0,E3 0.0,E4 0.0,E5 0.0,E6 0.0}
DECL FDAT FP16={TOOL_NO 5,BASE_NO 0,IPO_FRAME #BASE,POINT2[] " ",TQ_STATE FALSE}
DECL LDAT LCPDAT4={VEL 2.00000,ACC 100.000,APO_DIST 100.000,APO_FAC 50.0000,AXIS_VEL 100.000,AXIS_ACC 100.000,ORI_TYP #VAR,CIRC_TYP #BASE,JERK_FAC 50.0000,GEAR_JERK 50.0000,EXAX_IGN 0}
DECL E6POS XP17={X -1252.07056,Y -169.310532,Z 91.2468262,A -1.23850,B 1.32794106,C 179.761078,S 6,T 27,E1 0.0,E2 0.0,E3 0.0,E4 0.0,E5 0.0,E6 0.0}
DECL FDAT FP17={TOOL_NO 5,BASE_NO 0,IPO_FRAME #BASE,POINT2[] " ",TQ_STATE FALSE}
DECL LDAT LCPDAT5={VEL 2.00000,ACC 100.000,APO_DIST 100.000,APO_FAC 50.0000,AXIS_VEL 100.000,AXIS_ACC 100.000,ORI_TYP #VAR,CIRC_TYP #BASE,JERK_FAC 50.0000,GEAR_JERK 50.0000,EXAX_IGN 0}
DECL E6POS XP18={X -1252.07043,Y -169.310532,Z 1067.28162,A -1.23850,B 1.32794106,C 179.761078,S 6,T 27,E1 0.0,E2 0.0,E3 0.0,E4 0.0,E5 0.0,E6 0.0}
DECL FDAT FP18={TOOL_NO 5,BASE_NO 0,IPO_FRAME #BASE,POINT2[] " ",TQ_STATE FALSE}
DECL LDAT LCPDAT6={VEL 2.00000,ACC 100.000,APO_DIST 100.000,APO_FAC 50.0000,AXIS_VEL 100.000,AXIS_ACC 100.000,ORI_TYP #VAR,CIRC_TYP #BASE,JERK_FAC 50.0000,GEAR_JERK 50.0000,EXAX_IGN 0}
DECL E6POS XP19={X -905.921936,Y -172.186203,Z 2837.76685,A -5.97172117,B 82.0147247,C 174.335983,S 6,T 27,E1 0.0,E2 0.0,E3 0.0,E4 0.0,E5 0.0,E6 0.0}
DECL FDAT FP19={TOOL_NO 5,BASE_NO 0,IPO_FRAME #BASE,POINT2[] " ",TQ_STATE FALSE}
DECL PDAT PPDAT13={VEL 100.000,ACC 100.000,APO_DIST 100.000,APO_MODE #CDIS,GEAR_JERK 50.0000,EXAX_IGN 0}
ENDDAT
